SUBAPPLICATION Uebung_000b_AX (* AX_AND *)
  (* Standard: 61499-2; Description: Copyright (c) 2023 Meisterschulen am Ostbahnhof This program and the accompanying materials are made available under the terms of the Eclipse Public License 2.0 which is available at https://www.eclipse.org/legal/epl-2.0/ SPDX-License-Identifier: EPL-2.0 *)
  (* Version 1.0, 2026-01-16, Franz Höpfinger, Meisterschulen am Ostbahnhof, initial API and implementation and/or initial documentation *)
  PACKAGE Uebungen;
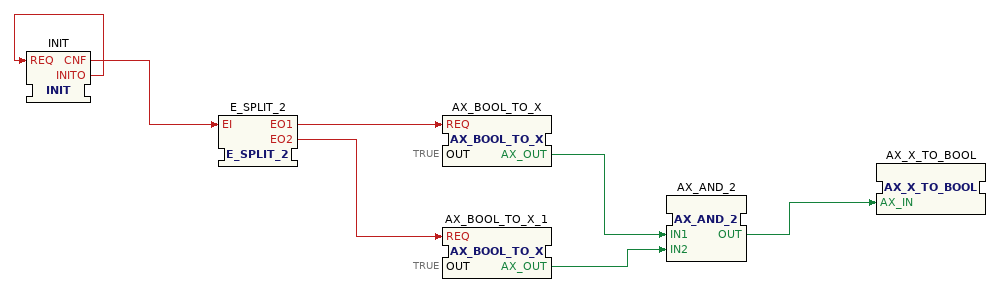
  FBS
    AX_AND_2 : adapter::booleanOperators::AX_AND_2;
    AX_X_TO_BOOL : adapter::conversion::unidirectional::AX_X_TO_BOOL;
    AX_BOOL_TO_X : adapter::conversion::unidirectional::AX_BOOL_TO_X(OUT := TRUE);
    AX_BOOL_TO_X_1 : adapter::conversion::unidirectional::AX_BOOL_TO_X(OUT := TRUE);
    INIT : iec61131::bitwiseOperators::INIT;
    E_SPLIT_2 : iec61499::events::E_SPLIT_2;
  END_FBS
  EVENT_CONNECTIONS
    INIT.CNF TO E_SPLIT_2.EI;
    E_SPLIT_2.EO1 TO AX_BOOL_TO_X.REQ;
    E_SPLIT_2.EO2 TO AX_BOOL_TO_X_1.REQ;
    INIT.INITO TO INIT.REQ;
  END_CONNECTIONS
  ADAPTER_CONNECTIONS
    AX_BOOL_TO_X.AX_OUT TO AX_AND_2.IN1;
    AX_BOOL_TO_X_1.AX_OUT TO AX_AND_2.IN2;
    AX_AND_2.OUT TO AX_X_TO_BOOL.AX_IN;
  END_CONNECTIONS
END_SUBAPPLICATION
